FUNCTION_BLOCK RecipeManager IMPLEMENTS Cyclic, Name
VAR
	values : ARRAY[0..RecipeParameters.ValueCountLimit - 1] OF RecipeValue;
	valueCount : INT;

	valueStringBuffer : STRING(RecipeParameters.TableBufferSize);
	_Buffer : STRING(RecipeParameters.BufferSize);
	sb : StringBuilderExtBuffer := (Buffer := ToAnyType(_Buffer));

	_FolderPath : T_MaxString;
	_FileName : T_MaxString;
	file : File;
	savingFile : BOOL;
	loadingFile : BOOL;
	directory : Directory;
	
	_JustLoaded : BOOL;
	_JustSaved : BOOL;

	_NewLine : STRING := '$N';
	_Assignment : STRING := ':=';
	_Extension : STRING := '.txt';
	_StringBoundary : STRING := '$'';
	
	_Name : T_MaxString;
	
	savedMessage : MessageEventLogger(TC_EVENTS.RecipeManagerEventClass.RecipeManagerSavedRecipe) := (Source := THIS^);
	loadedMessage : MessageEventLogger(TC_EVENTS.RecipeManagerEventClass.RecipeManagerLoadedRecipe) := (Source := THIS^);
END_VAR

METHOD AddSingleValue
VAR_INPUT
	value : ANY;
	name : T_MaxString;
END_VAR
VAR
	newValue : POINTER TO RecipeSingleValue;
END_VAR
IF (valueCount < RecipeParameters.ValueCountLimit) THEN
	newValue := __NEW(RecipeSingleValue);
	newValue^.Bind(value);
	newValue^.Name := name;
	newValue^.Assignment := _Assignment;
	values[valueCount] := newValue^;
	
	valueCount := valueCount + 1;
END_IF
END_METHOD

METHOD AddStringValue
VAR_INPUT
	value : ANY;
	name : T_MaxString;
END_VAR
VAR
	newValue : POINTER TO RecipeStringValue;
END_VAR
IF (valueCount < RecipeParameters.ValueCountLimit) THEN
	newValue := __NEW(RecipeStringValue);
	newValue^.Bind(value);
	newValue^.Buffer := ToAnyType(valueStringBuffer);
	newValue^.Name := name;
	newValue^.Assignment := _Assignment;
	values[valueCount] := newValue^;
	
	valueCount := valueCount + 1;
END_IF
END_METHOD

METHOD AddTableValue : REFERENCE TO RecipeTableValue
VAR_INPUT
	firstRow : ANY;
	name : T_MaxString;
END_VAR
VAR
	newValue : POINTER TO RecipeTableValue;
END_VAR
IF (valueCount < RecipeParameters.ValueCountLimit) THEN
	newValue := __NEW(RecipeTableValue);
	newValue^.Buffer := ToAnyType(valueStringBuffer);
	newValue^.DefineRow(firstRow);
	newValue^.Name := name;
	newValue^.Assignment := _Assignment;
	values[valueCount] := newValue^;
	
	valueCount := valueCount + 1;
	
	AddTableValue REF= newValue^;
END_IF
END_METHOD

{attribute 'monitoring' := 'call'}
PROPERTY Assignment : STRING
GET
Assignment := _Assignment;
END_GET
SET
_Assignment := Assignment;
END_SET
END_PROPERTY

PROPERTY BuildParseBuffer : REFERENCE TO StringBuilderExtBuffer
GET
BuildParseBuffer REF= sb;
END_GET
END_PROPERTY

METHOD BuildValueString : BOOL
VAR
	i : INT;
END_VAR
sb.Clear();
FOR i := 0 TO valueCount - 1 DO
	IF (i > 0) THEN
		sb.Append(_NewLine);
	END_IF
	sb.AppendByPointer(values[i].BuildAndGetAssignmentString());
END_FOR
END_METHOD

{attribute 'monitoring' := 'call'}
PROPERTY Busy : BOOL
GET
Busy := savingFile OR loadingFile;
END_GET
END_PROPERTY

METHOD Cyclic
file.Cyclic();
directory.Cyclic();

_JustSaved := FALSE;
_JustLoaded := FALSE;

IF (savingFile AND file.Done) THEN
	savingFile := FALSE;
	_JustSaved := TRUE;
	sb.Clear();
	ListRecipes();
	savedMessage.ClearArguments().AddStringByValue(_FileName);
	savedMessage.Send();
END_IF

IF (loadingFile AND file.Done) THEN
	loadingFile := FALSE;
	_JustLoaded := TRUE;
	ParseValueString();
	sb.Clear();
	loadedMessage.ClearArguments().AddStringByValue(_FileName);
	loadedMessage.Send();
END_IF

IF (NOT directory.ListDone) THEN
	ListRecipes();
END_IF
END_METHOD

{attribute 'monitoring' := 'call'}
PROPERTY Extension : STRING
GET
Extension := _Extension;
END_GET
SET
_Extension := Extension;
END_SET
END_PROPERTY

METHOD FB_exit : BOOL
VAR_INPUT
	bInCopyCode : BOOL; // if TRUE, the exit method is called for exiting an instance that is copied afterwards (online change).
END_VAR
VAR
	i : INT;
END_VAR
FOR i := 0 TO valueCount - 1 DO
	values[i].Dispose();
	values[i] := 0;
END_FOR
END_METHOD

METHOD FB_init : BOOL
VAR_INPUT
	bInitRetains : BOOL; // if TRUE, the retain variables are initialized (warm start / cold start)
	bInCopyCode : BOOL;  // if TRUE, the instance afterwards gets moved into the copy code (online change)
END_VAR
END_METHOD

{attribute 'monitoring' := 'call'}
PROPERTY FileName : T_MaxString
GET
FileName := _FileName;
END_GET
SET
_FileName := FileName;
END_SET
END_PROPERTY

{attribute 'monitoring' := 'call'}
PROPERTY FolderPath : T_MaxString
GET
FolderPath := _FolderPath;
END_GET
SET
_FolderPath := FolderPath;
END_SET
END_PROPERTY

METHOD PRIVATE GetRecipePath : T_MaxString
GetRecipePath := CONCAT(_FolderPath, _FileName);

IF (NOT StringEndsWithAny(_FileName, _Extension)) THEN
	GetRecipePath := CONCAT(GetRecipePath, _Extension);
END_IF
END_METHOD

METHOD GetTable : REFERENCE TO RecipeTableValue
VAR_INPUT
	name : T_MaxString;
END_VAR
VAR
	value : RecipeValue;
	p : POINTER TO RecipeTableValue;
END_VAR
value := GetValue(name);
__QUERYPOINTER(value, p);
IF (p <> 0) THEN
	GetTable REF= p^;
END_IF
END_METHOD

METHOD GetValue : RecipeValue
VAR_INPUT
	name : T_MaxString;
END_VAR
VAR
	i : INT;
END_VAR
FOR i := 0 TO valueCount - 1 DO
	IF (values[i].Name = name) THEN
		GetValue := values[i];
		RETURN;
	END_IF
END_FOR
END_METHOD

{attribute 'monitoring' := 'call'}
PROPERTY JustLoaded : BOOL
GET
JustLoaded := _JustLoaded;
END_GET
END_PROPERTY

{attribute 'monitoring' := 'call'}
PROPERTY JustSaved : BOOL
GET
JustSaved := _JustSaved;
END_GET
END_PROPERTY

{attribute 'monitoring' := 'call'}
PROPERTY ListLoaded : BOOL
GET
ListLoaded := directory.ListDone;
END_GET
END_PROPERTY

METHOD ListRecipes
VAR_INPUT
END_VAR
directory.List(
	BuildStringInline(_FolderPath)
		.Append('*')
		.Append(_Extension)
		.GetString()
);
END_METHOD

METHOD Load
IF (_FileName = '' OR _FolderPath = '') THEN
	RETURN;
END_IF

sb.Clear();

file.Read(
	buffer := ADR(_Buffer),
	bufferLength := SIZEOF(_Buffer) - 1,
	filePath := GetRecipePath()
);

loadingFile := TRUE;
END_METHOD

{attribute 'monitoring' := 'call'}
PROPERTY Name : T_MaxString
GET
Name := _Name;
END_GET
SET
_Name := Name;
END_SET
END_PROPERTY

{attribute 'monitoring' := 'call'}
PROPERTY NewLine : STRING
GET
NewLine := _NewLine;
END_GET
SET
_NewLine := NewLine;

//serializer.NewLine := _NewLine;
//deserializer.NewLine := _NewLine;
END_SET
END_PROPERTY

METHOD PRIVATE ParseValueString
VAR
	caret : DINT;
	assignmentLength : DINT;
	newLineLength : DINT;
	variableNameLength : DINT;
	variableName : T_MaxString;
	tableRowCountString : STRING;
	tableRowCount : INT;
	singleValueString : T_MaxString;
	valueLength : DINT;
	tableLineLength : DINT;
	newLineIndex : DINT;
	stringBoundaryLength : DINT;
	
	value : RecipeValue;
	singleValue : RecipeSingleValueType;
	stringValue : RecipeStringValueType;
	tableValue : RecipeTableValueType;
	
	sbValueBuffer : StringBuilderExtBuffer := (Buffer := ToAnyType(valueStringBuffer));

	i : INT;
END_VAR
sb.UpdateBufferLength();

assignmentLength := LEN(_Assignment);
newLineLength := LEN(_NewLine);
stringBoundaryLength := LEN(_StringBoundary);
WHILE caret < sb.Length DO
	// Search for assignment string
	variableNameLength := TO_DINT(FIND2(ADR(_Buffer[caret]), ADR(_Assignment))) - 1;
	IF (variableNameLength <= 0 OR variableNameLength > SIZEOF(T_MaxString) - 1) THEN
		EXIT;
	END_IF
	
	// Get variable name
	ClearData(variableName);
	SubString(_Buffer, variableName, caret, variableNameLength);
	variableName := F_LTrim(F_RTrim(variableName));
	tableRowCountString := F_LTrim(F_RTrim(GetStringBetween(variableName, '[', ']')));
	IF (LEN(tableRowCountString) > 0) THEN
		tableRowCount := STRING_TO_INT(tableRowCountString);
		variableName := LEFT(variableName, LEN(variableName) - LEN(tableRowCountString) - 2);
	ELSE
		tableRowCount := 0;
	END_IF
	
	caret := caret + variableNameLength + assignmentLength;
	
	// Find value by name
	value := GetValue(variableName);
	IF (value = 0) THEN
		CONTINUE;
	END_IF
	
	// Get value string
	// Parse and assign value
	// Update caret
	ClearData(singleValueString);
	IF (__QUERYINTERFACE(value, singleValue)) THEN
		valueLength := TO_DINT(FIND2(pSrcString := ADR(_Buffer[caret]), pFindString := ADR(_NewLine))) - 1;
		IF (valueLength < 0) THEN
			valueLength := sb.Length - caret;
		ELSIF (valueLength > SIZEOF(T_MaxString) - 1) THEN
			EXIT;
		END_IF
		SubString(_Buffer, singleValueString, caret, valueLength);
		singleValueString := F_LTrim(F_RTrim(singleValueString));
		singleValue.ParseAndAssignValue(singleValueString);
		caret := caret + valueLength + newLineLength;
	ELSIF (__QUERYINTERFACE(value, stringValue)) THEN
		caret := caret + TO_DINT(FIND2(
								pSrcString := ADR(_Buffer[caret]),
								pFindString := ADR(_StringBoundary)
						)) - 1 + stringBoundaryLength;
		valueLength := 0;
		WHILE TRUE DO
			valueLength := valueLength + TO_DINT(FIND2(
											pSrcString := ADR(_Buffer[caret + valueLength]),
											pFindString := ADR(_StringBoundary))
										) - 1;
			IF (valueLength = -1) THEN
				EXIT;
			ELSIF (caret + valueLength + 2 * stringBoundaryLength < sb.Length) THEN
				IF (StringBeginsWith(PSTRING_TO_STRING(ADR(_Buffer) + TO_DWORD(caret + valueLength + stringBoundaryLength)), _StringBoundary)) THEN
					valueLength := valueLength + 2 * stringBoundaryLength;
				ELSE 
					EXIT;
				END_IF 
			ELSE
				EXIT;
			END_IF
		END_WHILE
		sbValueBuffer.Clear().AppendSubString(_Buffer, caret, valueLength);
		stringValue.ParseAndAssignValue();
		newLineIndex := TO_DINT(FIND2(
									pSrcString := ADR(_Buffer[caret + valueLength + stringBoundaryLength]),
									pFindString := ADR(_NewLine)
							)) - 1;
		caret := caret + valueLength + stringBoundaryLength + newLineIndex + newLineLength;
	ELSIF (__QUERYINTERFACE(value, tableValue)) THEN
		FOR i := 0 TO 1 DO
			caret := caret + TO_DINT(FIND2(
									pSrcString := ADR(_Buffer[caret]),
									pFindString := ADR(_NewLine)
							)) - 1 + newLineLength;
		END_FOR
		valueLength := 0;
		FOR i := 0 TO tableRowCount - 1 DO
			tableLineLength := TO_DINT(FIND2(
									pSrcString := ADR(_Buffer[caret + valueLength]),
									pFindString := ADR(_NewLine)
							)) - 1 + newLineLength;
			IF (tableLineLength = 0) THEN
				tableLineLength := sb.Length - (caret + valueLength);
			END_IF
			valueLength := valueLength + tableLineLength;
		END_FOR
		sbValueBuffer.Clear().AppendSubString(_Buffer, caret, valueLength);
		tableValue.ParseAndAssignValues(tableRowCount);
		caret := caret + valueLength; // Newline is already included in table row search
	END_IF
END_WHILE
END_METHOD

METHOD RecipeExists : BOOL
VAR_INPUT
	name : T_MaxString;
END_VAR
VAR
	fileName : T_MaxString;
	i : INT;
	list : REFERENCE TO ARRAY[0..49] OF T_MaxString;
END_VAR
IF (name = '') THEN
	RETURN;
END_IF

IF (StringEndsWithAny(name, _Extension)) THEN
	fileName := name;
ELSE
	fileName := CONCAT(name, _Extension);
END_IF

list REF= RecipeList;
FOR i := 0 TO 49 DO
	IF (list[i] = '') THEN
		RETURN;
	END_IF
	IF (list[i] = fileName) THEN
		RecipeExists := TRUE;
		RETURN;
	END_IF
END_FOR
END_METHOD

{attribute 'monitoring' := 'call'}
PROPERTY RecipeList : REFERENCE TO ARRAY[0..49] OF T_MaxString
GET
RecipeList REF= directory.FileNameList;
END_GET
END_PROPERTY

METHOD Save
IF (_FileName = '' OR _FolderPath = '') THEN
	RETURN;
END_IF

BuildValueString();

file.Write(
	buffer := ADR(_Buffer),
	bufferLength := LEN2(ADR(_Buffer)),
	filePath := GetRecipePath(),
	append := FALSE
);

savingFile := TRUE;
END_METHOD

END_FUNCTION_BLOCK

(* stored: Version 1.1.0.1
   POU RecipeManager: Id {77c5c610-1c81-0616-06a3-6337e886bd1e}, SpecialFunc None
   Method AddSingleValue: Id {9c02c9fb-7c7b-0661-015f-e417480cf676}
   Method AddStringValue: Id {189baf3e-2ee6-0ea2-308a-17fa4409fecf}
   Method AddTableValue: Id {a0ec7a96-2cd5-06a8-338d-e79a080e8ef1}
   Property Assignment: Id {7b617ac0-6621-0620-25e6-167c8d314db3}
   Get Get: Id {ff7c6d30-30ed-05c0-15ed-a55cdafd19f5}
   Set Set: Id {b83d7434-de63-0421-248b-53035cc15ef9}
   Property BuildParseBuffer: Id {7764e3fa-19ce-0603-390f-e7376cb3160f}
   Get Get: Id {04b38d0d-2de1-0215-0560-02a87dcdea3e}
   Method BuildValueString: Id {f214b55b-5050-0596-38a7-7e0d32dc8021}
   Property Busy: Id {7cfa17eb-d3a3-07fa-3d85-776882933b67}
   Get Get: Id {99ff0090-9192-030e-0556-a7e5db2b7f61}
   Method Cyclic: Id {788b2b89-a987-0ac7-0a9d-51b6f200985e}
   Property Extension: Id {b2ad55aa-52f2-0956-066e-a1a2576c9f56}
   Get Get: Id {0e62e0c4-473c-0784-1ea5-a8f46398960e}
   Set Set: Id {bdd58266-6978-0f1a-2ec7-37de221f0f67}
   Method FB_exit: Id {eb111b38-3aef-0830-0bd7-caa81c03b2e3}
   Method FB_init: Id {8a42ac39-82f5-014b-0bba-01df588c4943}
   Property FileName: Id {122af664-9e40-0299-141f-ec89317ca077}
   Get Get: Id {d0dc6add-cd61-07c8-0a12-c52e0a4af129}
   Set Set: Id {6c1b1c2f-310a-01ed-009a-4841fd625cfb}
   Property FolderPath: Id {86b647fc-bf27-0419-0d76-a2f28385d87e}
   Get Get: Id {7e41cdcc-67a2-035c-364c-87055d04effd}
   Set Set: Id {4581bd7b-a2f8-0080-3203-1c1a2fa0e72e}
   Method GetRecipePath: Id {aa927626-c3f3-0065-0867-fe8915b16b40}
   Method GetTable: Id {ebd01b12-3e62-008e-1e08-da5f95dc4ad3}
   Method GetValue: Id {bb49e33a-de77-0d8c-1bfc-e271c4ee3ff5}
   Property JustLoaded: Id {2077e4de-4c40-0aeb-0b63-275e0632eaf0}
   Get Get: Id {dbfa9129-0a70-0d56-33d3-bb4fc63f0d3d}
   Property JustSaved: Id {35c04087-3a17-0a9a-36f5-3fc152d5e4f8}
   Get Get: Id {75ffa0b7-f455-05fe-1195-95f3478693dc}
   Property ListLoaded: Id {56b2a616-06f4-01b1-10be-4d33872b8012}
   Get Get: Id {0718b734-43a3-0db1-36cd-88083ba12ec5}
   Method ListRecipes: Id {06b24d78-54a3-0fd9-025f-f678dfd8873d}
   Method Load: Id {e13ba227-265c-003c-16a9-027fd14cba33}
   Property Name: Id {01bb3166-5490-0205-2121-3fe3bb87d958}
   Get Get: Id {0dacc52b-4c63-03e6-08ca-dc2fabd0f5cb}
   Set Set: Id {c104e843-fcb5-02c5-00b8-f062a5fd3fb3}
   Property NewLine: Id {5e9e4f96-dcb0-0eff-0f4b-96624bfd49c8}
   Get Get: Id {a0908233-b4ff-0b65-14b9-2990cbb2630f}
   Set Set: Id {8e433a38-c0cb-0c47-2e09-30d231261540}
   Method ParseValueString: Id {f8989f6e-d562-0c64-0845-3edcee6fa0d9}
   Method RecipeExists: Id {362dcd42-3486-0c62-11af-643746cf951e}
   Property RecipeList: Id {53671a00-5ebb-040a-0250-856488ee25e9}
   Get Get: Id {cc34b112-61db-075c-07c4-6224ca7c3cef}
   Method Save: Id {f0759a7e-99b2-0933-354d-07d2436af8d4} *)
